Universal Robots PolyScope program: proiectfinal.urp

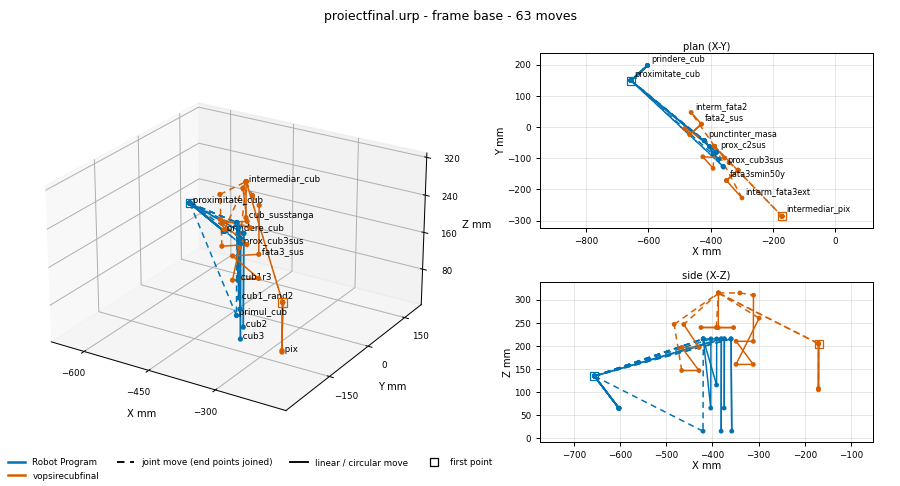
[picture p0: tool path of proiectfinal.urp in frame base, 63 of 63 moves have a stored position in this frame; points joined in program order, loops and branches not executed]
Program testproiectfinal2 (installation=default directory=/programs/usbdisk/final createdIn=3.15.5.106321 lastSavedIn=3.15.6.106324 robotSerialNumber=2021351072)
Calibrated DH parameters: a=[0.000146, -0.006215, -0.392465, 0.000066, 0.00001, 0]; d=[0.089346, 308.112025, -307.666795, -0.334946, 0.094852, 0.082573]; alpha=[1.570365, -0.001381, 0.017393, 1.570287, -1.570555, 0]; deltaTheta=[0.000031, -1.556209, 1.575918, -0.019781, 0.000038, 0.000088]
Robot Program (runOnlyOnce=false)
  MoveJ speed 60 deg/s, acceleration 80 deg/s^2 (useActiveTCP=false) tcp=Palet
    Waypoint proximitate_cub: TCP in base x=-655.658 y=149.782 z=135.002 mm, rx=1.0761 ry=2.3886 rz=1.0065 rad; joints [-7.715, -31.545, 17.047, -40.87, -122.454, -38.841] deg; flange x=-782.032 y=40.366 z=298.765 mm, rx=1.0761 ry=2.3886 rz=1.0065 rad
  MoveL speed 250 mm/s, acceleration 1200 mm/s^2 (useActiveTCP=true) feature=Base
    Waypoint prindere_cub: TCP in base x=-602.576 y=198.07 z=65.356 mm, rx=1.0761 ry=2.3886 rz=1.0065 rad; joints [-11.8, -45.21, 53.1, -65.52, -124.71, -42.93] deg; flange x=-728.95 y=88.654 z=229.118 mm, rx=1.0761 ry=2.3886 rz=1.0065 rad
    Wait Sleep waitTime=0.5
    'G40'
    URCap RG Grip (OnRobot, OnRobot A/S) dataModel(rg-target-force=40.0, rg-target-width=0.04, Variable(key=on_return, variable(name=on_return)))
  MoveL speed 250 mm/s, acceleration 1200 mm/s^2 (useActiveTCP=true) feature=Base
    Waypoint proximitate_cub: TCP in base x=-655.658 y=149.782 z=135.002 mm, rx=1.0761 ry=2.3886 rz=1.0065 rad; joints [-7.715, -31.545, 17.047, -40.87, -122.454, -38.841] deg; flange x=-782.032 y=40.366 z=298.765 mm, rx=1.0761 ry=2.3886 rz=1.0065 rad
  MoveJ speed 60 deg/s, acceleration 80 deg/s^2 (useActiveTCP=true)
    Waypoint punctinter_masa: TCP in base x=-419.876 y=-42.977 z=215.649 mm, rx=2.9437 ry=1.0488 rz=-0.0163 rad; joints [-9.726, -100.905, 97.2, -86.353, -88.88, 41.054] deg; flange x=-418.643 y=-40.621 z=449.643 mm, rx=2.9437 ry=1.0488 rz=-0.0163 rad
  MoveJ speed 60 deg/s, acceleration 80 deg/s^2 (useActiveTCP=true)
    Waypoint primul_cub: TCP in base x=-420.36 y=-43.654 z=15.65 mm, rx=2.9437 ry=1.0488 rz=-0.0163 rad; joints [-9.62, -94.93, 122.37, -117.5, -88.88, 41.16] deg; flange x=-419.127 y=-41.298 z=249.645 mm, rx=2.9437 ry=1.0488 rz=-0.0163 rad
    Wait Sleep waitTime=0.5
    'G80'
    URCap RG Grip (OnRobot, OnRobot A/S) dataModel(rg-target-force=40.0, rg-target-width=0.08)
  MoveJ speed 60 deg/s, acceleration 80 deg/s^2 (useActiveTCP=true)
    Waypoint proximitate_cub: TCP in base x=-655.658 y=149.782 z=135.002 mm, rx=1.0761 ry=2.3886 rz=1.0065 rad; joints [-7.715, -31.545, 17.047, -40.87, -122.454, -38.841] deg; flange x=-782.032 y=40.366 z=298.765 mm, rx=1.0761 ry=2.3886 rz=1.0065 rad
  MoveL speed 250 mm/s, acceleration 1200 mm/s^2 (useActiveTCP=true) feature=Base
    Waypoint prindere_cub: TCP in base x=-602.576 y=198.07 z=65.356 mm, rx=1.0761 ry=2.3886 rz=1.0065 rad; joints [-11.8, -45.21, 53.1, -65.52, -124.71, -42.93] deg; flange x=-728.95 y=88.654 z=229.118 mm, rx=1.0761 ry=2.3886 rz=1.0065 rad
    Wait Sleep waitTime=0.5
    'G40'
    URCap RG Grip (OnRobot, OnRobot A/S) dataModel(rg-target-force=40.0, rg-target-width=0.04)
  MoveJ speed 60 deg/s, acceleration 80 deg/s^2 (useActiveTCP=true)
    Waypoint proximitate_cub: TCP in base x=-655.658 y=149.782 z=135.002 mm, rx=1.0761 ry=2.3886 rz=1.0065 rad; joints [-7.715, -31.545, 17.047, -40.87, -122.454, -38.841] deg; flange x=-782.032 y=40.366 z=298.765 mm, rx=1.0761 ry=2.3886 rz=1.0065 rad
  MoveL speed 250 mm/s, acceleration 1200 mm/s^2 (useActiveTCP=true) feature=Base
    Waypoint prox_c2sus: TCP in base x=-380.694 y=-80.38 z=215.695 mm, rx=2.9437 ry=1.0488 rz=-0.0163 rad; joints [-4.992, -105.625, 100.759, -85.284, -88.888, 45.789] deg; flange x=-379.461 y=-78.023 z=449.69 mm, rx=2.9437 ry=1.0488 rz=-0.0163 rad
  MoveL speed 250 mm/s, acceleration 1200 mm/s^2 (useActiveTCP=true) feature=Base
    Waypoint cub2: TCP in base x=-381.178 y=-81.057 z=15.697 mm, rx=2.9437 ry=1.0488 rz=-0.0163 rad; joints [-4.881, -99.963, 126.628, -116.816, -88.889, 45.899] deg; flange x=-379.945 y=-78.7 z=249.691 mm, rx=2.9437 ry=1.0488 rz=-0.0163 rad
    Wait Sleep waitTime=0.5
    'G80'
    URCap RG Grip (OnRobot, OnRobot A/S) dataModel(rg-target-force=40.0, rg-target-width=0.08)
  MoveL speed 250 mm/s, acceleration 1200 mm/s^2 (useActiveTCP=true) feature=Base
    Waypoint prox_cub2: TCP in base x=-380.694 y=-80.38 z=215.695 mm, rx=2.9437 ry=1.0488 rz=-0.0163 rad; joints [-4.992, -105.625, 100.759, -85.284, -88.888, 45.789] deg; flange x=-379.461 y=-78.023 z=449.69 mm, rx=2.9437 ry=1.0488 rz=-0.0163 rad
  MoveJ speed 60 deg/s, acceleration 80 deg/s^2 (useActiveTCP=true)
    Waypoint proximitate_cub: TCP in base x=-655.658 y=149.782 z=135.002 mm, rx=1.0761 ry=2.3886 rz=1.0065 rad; joints [-7.715, -31.545, 17.047, -40.87, -122.454, -38.841] deg; flange x=-782.032 y=40.366 z=298.765 mm, rx=1.0761 ry=2.3886 rz=1.0065 rad
  MoveL speed 250 mm/s, acceleration 1200 mm/s^2 (useActiveTCP=true) feature=Base
    Waypoint prindere_cub: TCP in base x=-602.576 y=198.07 z=65.356 mm, rx=1.0761 ry=2.3886 rz=1.0065 rad; joints [-11.8, -45.21, 53.1, -65.52, -124.71, -42.93] deg; flange x=-728.95 y=88.654 z=229.118 mm, rx=1.0761 ry=2.3886 rz=1.0065 rad
    Wait Sleep waitTime=0.5
    'G40'
    URCap RG Grip (OnRobot, OnRobot A/S) dataModel(rg-target-force=40.0, rg-target-width=0.04)
  MoveJ speed 60 deg/s, acceleration 80 deg/s^2 (useActiveTCP=true)
    Waypoint proximitate_cub: TCP in base x=-655.658 y=149.782 z=135.002 mm, rx=1.0761 ry=2.3886 rz=1.0065 rad; joints [-7.715, -31.545, 17.047, -40.87, -122.454, -38.841] deg; flange x=-782.032 y=40.366 z=298.765 mm, rx=1.0761 ry=2.3886 rz=1.0065 rad
  MoveJ speed 60 deg/s, acceleration 80 deg/s^2 (useActiveTCP=true)
    Waypoint prox_cub3sus: TCP in base x=-359.676 y=-125.655 z=215.741 mm, rx=2.9437 ry=1.0488 rz=-0.0163 rad; joints [2.001, -106.845, 101.634, -85.073, -88.915, 52.783] deg; flange x=-358.443 y=-123.298 z=449.736 mm, rx=2.9437 ry=1.0488 rz=-0.0163 rad
  MoveL speed 250 mm/s, acceleration 1200 mm/s^2 (useActiveTCP=true) feature=Base
    Waypoint cub3: TCP in base x=-358.165 y=-128.509 z=15.708 mm, rx=2.9439 ry=1.0486 rz=-0.0162 rad; joints [2.174, -101.579, 127.644, -116.344, -87.985, 53.434] deg; flange x=-356.947 y=-126.168 z=249.703 mm, rx=2.9439 ry=1.0486 rz=-0.0162 rad
    Wait Sleep waitTime=0.5
    'G80'
    URCap RG Grip (OnRobot, OnRobot A/S) dataModel(rg-target-force=40.0, rg-target-width=0.08)
  MoveL speed 250 mm/s, acceleration 1200 mm/s^2 (useActiveTCP=true) feature=Base
    Waypoint prox_cub3: TCP in base x=-359.676 y=-125.655 z=215.741 mm, rx=2.9437 ry=1.0488 rz=-0.0163 rad; joints [2.001, -106.845, 101.634, -85.073, -88.915, 52.783] deg; flange x=-358.443 y=-123.298 z=449.736 mm, rx=2.9437 ry=1.0488 rz=-0.0163 rad
  MoveJ speed 60 deg/s, acceleration 80 deg/s^2 (useActiveTCP=true)
    Waypoint proximitate_cub: TCP in base x=-655.658 y=149.782 z=135.002 mm, rx=1.0761 ry=2.3886 rz=1.0065 rad; joints [-7.715, -31.545, 17.047, -40.87, -122.454, -38.841] deg; flange x=-782.032 y=40.366 z=298.765 mm, rx=1.0761 ry=2.3886 rz=1.0065 rad
  MoveL speed 250 mm/s, acceleration 1200 mm/s^2 (useActiveTCP=true) feature=Base
    Waypoint prindere_cub: TCP in base x=-602.576 y=198.07 z=65.356 mm, rx=1.0761 ry=2.3886 rz=1.0065 rad; joints [-11.8, -45.21, 53.1, -65.52, -124.71, -42.93] deg; flange x=-728.95 y=88.654 z=229.118 mm, rx=1.0761 ry=2.3886 rz=1.0065 rad
    Wait Sleep waitTime=0.5
    'G40'
    URCap RG Grip (OnRobot, OnRobot A/S) dataModel(rg-target-force=40.0, rg-target-width=0.04)
  MoveL speed 250 mm/s, acceleration 1200 mm/s^2 (useActiveTCP=true) feature=Base
    Waypoint proximitate_cub: TCP in base x=-655.658 y=149.782 z=135.002 mm, rx=1.0761 ry=2.3886 rz=1.0065 rad; joints [-7.715, -31.545, 17.047, -40.87, -122.454, -38.841] deg; flange x=-782.032 y=40.366 z=298.765 mm, rx=1.0761 ry=2.3886 rz=1.0065 rad
  MoveJ speed 60 deg/s, acceleration 80 deg/s^2 (useActiveTCP=true)
    Waypoint punctinter_masa: TCP in base x=-419.876 y=-42.977 z=215.649 mm, rx=2.9437 ry=1.0488 rz=-0.0163 rad; joints [-9.726, -100.905, 97.2, -86.353, -88.88, 41.054] deg; flange x=-418.643 y=-40.621 z=449.643 mm, rx=2.9437 ry=1.0488 rz=-0.0163 rad
  MoveL speed 250 mm/s, acceleration 1200 mm/s^2 (useActiveTCP=true) feature=Base
    Waypoint cub1_rand2: TCP in base x=-403.648 y=-62.186 z=65.673 mm, rx=2.9437 ry=1.0488 rz=-0.0163 rad; joints [-7.34, -100.148, 118.843, -108.8, -88.883, 43.44] deg; flange x=-402.415 y=-59.83 z=299.668 mm, rx=2.9437 ry=1.0488 rz=-0.0163 rad
    Wait Sleep waitTime=0.5
    'G80'
    URCap RG Grip (OnRobot, OnRobot A/S) dataModel(rg-target-force=40.0, rg-target-width=0.08)
  MoveL speed 250 mm/s, acceleration 1200 mm/s^2 (useActiveTCP=true) feature=Base
    Waypoint ridicare_cub1r2: TCP in base x=-403.285 y=-61.678 z=215.672 mm, rx=2.9437 ry=1.0488 rz=-0.0163 rad; joints [-7.421, -102.916, 98.768, -85.955, -88.883, 43.359] deg; flange x=-402.052 y=-59.322 z=449.667 mm, rx=2.9437 ry=1.0488 rz=-0.0163 rad
  MoveJ speed 60 deg/s, acceleration 80 deg/s^2 (useActiveTCP=true)
    Waypoint proximitate_cub: TCP in base x=-655.658 y=149.782 z=135.002 mm, rx=1.0761 ry=2.3886 rz=1.0065 rad; joints [-7.715, -31.545, 17.047, -40.87, -122.454, -38.841] deg; flange x=-782.032 y=40.366 z=298.765 mm, rx=1.0761 ry=2.3886 rz=1.0065 rad
  MoveL speed 250 mm/s, acceleration 1200 mm/s^2 (useActiveTCP=true) feature=Base
    Waypoint prindere_cub: TCP in base x=-602.576 y=198.07 z=65.356 mm, rx=1.0761 ry=2.3886 rz=1.0065 rad; joints [-11.8, -45.21, 53.1, -65.52, -124.71, -42.93] deg; flange x=-728.95 y=88.654 z=229.118 mm, rx=1.0761 ry=2.3886 rz=1.0065 rad
    Wait Sleep waitTime=0.5
    'G40'
    URCap RG Grip (OnRobot, OnRobot A/S) dataModel(rg-target-force=40.0, rg-target-width=0.04)
  MoveL speed 250 mm/s, acceleration 1200 mm/s^2 (useActiveTCP=true) feature=Base
    Waypoint proximitate_cub: TCP in base x=-655.658 y=149.782 z=135.002 mm, rx=1.0761 ry=2.3886 rz=1.0065 rad; joints [-7.715, -31.545, 17.047, -40.87, -122.454, -38.841] deg; flange x=-782.032 y=40.366 z=298.765 mm, rx=1.0761 ry=2.3886 rz=1.0065 rad
  MoveJ speed 60 deg/s, acceleration 80 deg/s^2 (useActiveTCP=true)
    Waypoint punctinter_masa: TCP in base x=-419.876 y=-42.977 z=215.649 mm, rx=2.9437 ry=1.0488 rz=-0.0163 rad; joints [-9.726, -100.905, 97.2, -86.353, -88.88, 41.054] deg; flange x=-418.643 y=-40.621 z=449.643 mm, rx=2.9437 ry=1.0488 rz=-0.0163 rad
  MoveL speed 250 mm/s, acceleration 1200 mm/s^2 (useActiveTCP=true) feature=Base
    Waypoint prox_c2r2sus: TCP in base x=-374.19 y=-103.473 z=215.718 mm, rx=2.9437 ry=1.0488 rz=-0.0163 rad; joints [-1.482, -105.778, 100.88, -85.32, -88.9, 49.299] deg; flange x=-372.957 y=-101.117 z=449.713 mm, rx=2.9437 ry=1.0488 rz=-0.0163 rad
  MoveL speed 250 mm/s, acceleration 1200 mm/s^2 (useActiveTCP=true) feature=Base
    Waypoint cub2_r2: TCP in base x=-374.553 y=-103.981 z=65.719 mm, rx=2.9437 ry=1.0488 rz=-0.0163 rad; joints [-1.402, -103.233, 121.237, -108.224, -88.9, 49.379] deg; flange x=-373.321 y=-101.625 z=299.714 mm, rx=2.9437 ry=1.0488 rz=-0.0163 rad
    Wait Sleep waitTime=0.5
    'G80'
    URCap RG Grip (OnRobot, OnRobot A/S) dataModel(rg-target-force=40.0, rg-target-width=0.08)
  MoveL speed 250 mm/s, acceleration 1200 mm/s^2 (useActiveTCP=true) feature=Base
    Waypoint prox_cub2r2: TCP in base x=-374.19 y=-103.473 z=215.718 mm, rx=2.9437 ry=1.0488 rz=-0.0163 rad; joints [-1.482, -105.778, 100.88, -85.32, -88.9, 49.299] deg; flange x=-372.958 y=-101.117 z=449.713 mm, rx=2.9437 ry=1.0488 rz=-0.0163 rad
  MoveJ speed 60 deg/s, acceleration 80 deg/s^2 (useActiveTCP=true)
    Waypoint proximitate_cub: TCP in base x=-655.658 y=149.782 z=135.002 mm, rx=1.0761 ry=2.3886 rz=1.0065 rad; joints [-7.715, -31.545, 17.047, -40.87, -122.454, -38.841] deg; flange x=-782.032 y=40.366 z=298.765 mm, rx=1.0761 ry=2.3886 rz=1.0065 rad
  MoveL speed 250 mm/s, acceleration 1200 mm/s^2 (useActiveTCP=true) feature=Base
    Waypoint prindere_cub: TCP in base x=-602.576 y=198.07 z=65.356 mm, rx=1.0761 ry=2.3886 rz=1.0065 rad; joints [-11.8, -45.21, 53.1, -65.52, -124.71, -42.93] deg; flange x=-728.95 y=88.654 z=229.118 mm, rx=1.0761 ry=2.3886 rz=1.0065 rad
    Wait Sleep waitTime=0.5
    'G40'
    URCap RG Grip (OnRobot, OnRobot A/S) dataModel(rg-target-force=40.0, rg-target-width=0.04)
  MoveL speed 250 mm/s, acceleration 1200 mm/s^2 (useActiveTCP=true) feature=Base
    Waypoint proximitate_cub: TCP in base x=-655.658 y=149.782 z=135.002 mm, rx=1.0761 ry=2.3886 rz=1.0065 rad; joints [-7.715, -31.545, 17.047, -40.87, -122.454, -38.841] deg; flange x=-782.032 y=40.366 z=298.765 mm, rx=1.0761 ry=2.3886 rz=1.0065 rad
  MoveJ speed 60 deg/s, acceleration 80 deg/s^2 (useActiveTCP=true)
    Waypoint punctinter_masa: TCP in base x=-419.876 y=-42.977 z=215.649 mm, rx=2.9437 ry=1.0488 rz=-0.0163 rad; joints [-9.726, -100.905, 97.2, -86.353, -88.88, 41.054] deg; flange x=-418.643 y=-40.621 z=449.643 mm, rx=2.9437 ry=1.0488 rz=-0.0163 rad
  MoveL speed 250 mm/s, acceleration 1200 mm/s^2 (useActiveTCP=true) feature=Base
    Waypoint cub1r3: TCP in base x=-391.023 y=-85.111 z=115.696 mm, rx=2.9437 ry=1.0488 rz=-0.0163 rad; joints [-4.15, -103.314, 113.748, -100.6, -88.891, 46.631] deg; flange x=-389.79 y=-82.754 z=349.691 mm, rx=2.9437 ry=1.0488 rz=-0.0163 rad
    Wait Sleep waitTime=0.5
    'G80'
    URCap RG Grip (OnRobot, OnRobot A/S) dataModel(rg-target-force=40.0, rg-target-width=0.08)
  MoveL speed 250 mm/s, acceleration 1200 mm/s^2 (useActiveTCP=true) feature=Base
    Waypoint prox_c3r3s: TCP in base x=-390.781 y=-84.772 z=215.695 mm, rx=2.9437 ry=1.0488 rz=-0.0163 rad; joints [-4.203, -104.095, 99.659, -85.73, -88.891, 46.578] deg; flange x=-389.548 y=-82.415 z=449.69 mm, rx=2.9437 ry=1.0488 rz=-0.0163 rad
  Call vopsirecubfinal
SubProgram -> vopsirecubfinal
SubProgram vopsirecubfinal (keepSynchronizedWithDisk=false) programFile=/home/ur/ursim-current/programs/vopsirecubfinal.urp
  MoveJ speed 60 deg/s, acceleration 80 deg/s^2 (useActiveTCP=true)
    Waypoint intermediar_pix: TCP in base x=-170.071 y=-286.315 z=205.284 mm, rx=1.291 ry=2.848 rz=-0.0146 rad; joints [39.36, -114.129, 107.637, -83.618, -89.01, -1.87] deg; flange x=-170.186 y=-282.604 z=439.264 mm, rx=1.291 ry=2.848 rz=-0.0146 rad
  MoveL speed 250 mm/s, acceleration 1200 mm/s^2 (useActiveTCP=true) feature=Base
    Waypoint pix: TCP in base x=-170.313 y=-286.653 z=105.285 mm, rx=1.291 ry=2.848 rz=-0.0146 rad; joints [39.38, -113.83, 122.12, -98.4, -89.01, -1.85] deg; flange x=-170.428 y=-282.942 z=339.265 mm, rx=1.291 ry=2.848 rz=-0.0146 rad
    Wait Sleep waitTime=0.5
    URCap RG Grip (OnRobot, OnRobot A/S) dataModel(rg-target-force=40.0, rg-target-width=0.01)
    'G10'
  MoveJ speed 60 deg/s, acceleration 80 deg/s^2 (useActiveTCP=true)
    Waypoint intermediar_pix: TCP in base x=-170.071 y=-286.315 z=205.284 mm, rx=1.291 ry=2.848 rz=-0.0146 rad; joints [39.36, -114.129, 107.637, -83.618, -89.01, -1.87] deg; flange x=-170.186 y=-282.604 z=439.264 mm, rx=1.291 ry=2.848 rz=-0.0146 rad
  MoveJ speed 60 deg/s, acceleration 80 deg/s^2 (useActiveTCP=true)
    Waypoint intermediar_cub: TCP in base x=-387.106 y=-61.589 z=315.134 mm, rx=1.2835 ry=2.8619 rz=-0.034 rad; joints [-8.293, -102.753, 83.777, -71.093, -88.73, -49.983] deg; flange x=-383.978 y=-56.18 z=549.06 mm, rx=1.2835 ry=2.8619 rz=-0.034 rad
  MoveL speed 250 mm/s, acceleration 1200 mm/s^2 (useActiveTCP=true) feature=Base
    Waypoint cub_susstanga: TCP in base x=-387.287 y=-61.843 z=240.134 mm, rx=1.2835 ry=2.8619 rz=-0.034 rad; joints [-8.25, -105.11, 96.79, -81.75, -88.73, -49.94] deg; flange x=-384.16 y=-56.434 z=474.061 mm, rx=1.2835 ry=2.8619 rz=-0.034 rad
  MoveL speed 250 mm/s, acceleration 1200 mm/s^2 (useActiveTCP=true) feature=Base
    Waypoint cub_susdreapta: TCP in base x=-354.105 y=-99.246 z=240.181 mm, rx=1.2835 ry=2.8619 rz=-0.034 rad; joints [-2.814, -108.653, 99.227, -80.764, -88.742, -44.503] deg; flange x=-350.978 y=-93.837 z=474.107 mm, rx=1.2835 ry=2.8619 rz=-0.034 rad
  MoveL speed 250 mm/s, acceleration 1200 mm/s^2 (useActiveTCP=true) feature=Base
    Waypoint diagstangjos: TCP in base x=-424.69 y=-95.025 z=240.337 mm, rx=1.2835 ry=2.8619 rz=-0.034 rad; joints [-2.918, -99.183, 92.225, -83.229, -88.742, -44.606] deg; flange x=-421.562 y=-89.615 z=474.264 mm, rx=1.2835 ry=2.8619 rz=-0.034 rad
  MoveL speed 250 mm/s, acceleration 1200 mm/s^2 (useActiveTCP=true) feature=Base
    Waypoint cub_dreaptajos: TCP in base x=-391.508 y=-132.427 z=240.384 mm, rx=1.2835 ry=2.8619 rz=-0.034 rad; joints [2.359, -102.313, 94.738, -82.728, -88.765, -39.328] deg; flange x=-388.38 y=-127.018 z=474.31 mm, rx=1.2835 ry=2.8619 rz=-0.034 rad
  MoveJ speed 60 deg/s, acceleration 80 deg/s^2 (useActiveTCP=true)
    Waypoint intermediar_cub: TCP in base x=-387.106 y=-61.589 z=315.134 mm, rx=1.2835 ry=2.8619 rz=-0.034 rad; joints [-8.293, -102.753, 83.777, -71.093, -88.73, -49.983] deg; flange x=-383.978 y=-56.18 z=549.06 mm, rx=1.2835 ry=2.8619 rz=-0.034 rad
  MoveJ speed 60 deg/s, acceleration 80 deg/s^2 (useActiveTCP=true)
    Waypoint interm_latdrcub: TCP in base x=-340.651 y=-113.953 z=315.198 mm, rx=1.2835 ry=2.8619 rz=-0.034 rad; joints [-0.408, -107.27, 86.983, -69.955, -88.751, -42.096] deg; flange x=-337.523 y=-108.544 z=549.125 mm, rx=1.2835 ry=2.8619 rz=-0.034 rad
  MoveJ speed 60 deg/s, acceleration 80 deg/s^2 (useActiveTCP=true)
    Waypoint interm_fata3: TCP in base x=-311.097 y=-137.967 z=310.289 mm, rx=-0.1394 ry=-2.5859 rz=-0.5323 rad; joints [36.655, -116.066, 104.459, -87.091, -125.726, -49.98] deg; flange x=-205.123 y=-228.798 z=498.118 mm, rx=-0.1394 ry=-2.5859 rz=-0.5323 rad
  MoveL speed 250 mm/s, acceleration 1200 mm/s^2 (useActiveTCP=true) feature=Base
    Waypoint fata3_sus: TCP in base x=-311.331 y=-138.32 z=210.278 mm, rx=-0.1394 ry=-2.586 rz=-0.5323 rad; joints [36.68, -117.15, 119.7, -101.23, -125.726, -49.95] deg; flange x=-205.363 y=-229.14 z=398.116 mm, rx=-0.1394 ry=-2.586 rz=-0.5323 rad
  MoveL speed 250 mm/s, acceleration 1200 mm/s^2 (useActiveTCP=true) feature=Base
    Waypoint fata3smin50y: TCP in base x=-348.733 y=-171.502 z=210.481 mm, rx=-0.1394 ry=-2.586 rz=-0.5323 rad; joints [37.395, -109.418, 115.134, -103.887, -125.831, -49.078] deg; flange x=-242.766 y=-262.322 z=398.319 mm, rx=-0.1394 ry=-2.586 rz=-0.5323 rad
  MoveL speed 250 mm/s, acceleration 1200 mm/s^2 (useActiveTCP=true) feature=Base
    Waypoint diag: TCP in base x=-311.452 y=-138.489 z=160.278 mm, rx=-0.1394 ry=-2.586 rz=-0.5323 rad; joints [36.692, -116.21, 126.574, -109.035, -125.728, -49.935] deg; flange x=-205.484 y=-229.309 z=348.116 mm, rx=-0.1394 ry=-2.586 rz=-0.5323 rad
  MoveL speed 250 mm/s, acceleration 1200 mm/s^2 (useActiveTCP=true) feature=Base
    Waypoint fata3josmin50y: TCP in base x=-348.854 y=-171.671 z=160.481 mm, rx=-0.1394 ry=-2.586 rz=-0.5323 rad; joints [37.405, -108.1, 121.695, -111.758, -125.832, -49.066] deg; flange x=-242.887 y=-262.491 z=348.319 mm, rx=-0.1394 ry=-2.586 rz=-0.5323 rad
  MoveL speed 250 mm/s, acceleration 1200 mm/s^2 (useActiveTCP=true) feature=Base
    Waypoint interm_fata3ext: TCP in base x=-298.839 y=-227.436 z=260.55 mm, rx=-0.1394 ry=-2.586 rz=-0.5323 rad; joints [49.496, -106.173, 103.501, -86.61, -126.623, -34.094] deg; flange x=-192.872 y=-318.256 z=448.388 mm, rx=-0.1394 ry=-2.586 rz=-0.5323 rad
  MoveJ speed 60 deg/s, acceleration 80 deg/s^2 (useActiveTCP=true)
    Waypoint intermediar_cub: TCP in base x=-387.106 y=-61.589 z=315.134 mm, rx=1.2835 ry=2.8619 rz=-0.034 rad; joints [-8.293, -102.753, 83.777, -71.093, -88.73, -49.983] deg; flange x=-383.978 y=-56.18 z=549.06 mm, rx=1.2835 ry=2.8619 rz=-0.034 rad
  MoveJ speed 60 deg/s, acceleration 80 deg/s^2 (useActiveTCP=true)
    Waypoint interm_fata2: TCP in base x=-462.134 y=47.249 z=246.923 mm, rx=1.5541 ry=1.7177 rz=-0.4294 rad; joints [-35.631, -69.065, 63.951, -39.612, -67.495, -50.842] deg; flange x=-533.143 y=209.077 z=400.318 mm, rx=1.5541 ry=1.7177 rz=-0.4294 rad
  MoveL speed 250 mm/s, acceleration 1200 mm/s^2 (useActiveTCP=true) feature=Base
    Waypoint fata2_sus: TCP in base x=-429.073 y=9.677 z=196.969 mm, rx=1.5541 ry=1.7177 rz=-0.4294 rad; joints [-34.48, -75.75, 80.19, -49.51, -66.68, -49.96] deg; flange x=-500.082 y=171.505 z=350.364 mm, rx=1.5541 ry=1.7177 rz=-0.4294 rad
  MoveL speed 250 mm/s, acceleration 1200 mm/s^2 (useActiveTCP=true) feature=Base
    Waypoint fata2susmin50y: TCP in base x=-466.475 y=-23.504 z=197.172 mm, rx=1.5541 ry=1.7177 rz=-0.4294 rad; joints [-29.692, -72.801, 76.621, -50.493, -63.345, -46.169] deg; flange x=-537.484 y=138.324 z=350.567 mm, rx=1.5541 ry=1.7177 rz=-0.4294 rad
  MoveL speed 250 mm/s, acceleration 1200 mm/s^2 (useActiveTCP=true) feature=Base
    Waypoint diag2: TCP in base x=-429.194 y=9.508 z=146.97 mm, rx=1.5541 ry=1.7177 rz=-0.4294 rad; joints [-34.459, -74.801, 86.357, -56.633, -66.665, -49.944] deg; flange x=-500.203 y=171.336 z=300.365 mm, rx=1.5541 ry=1.7177 rz=-0.4294 rad
  MoveL speed 250 mm/s, acceleration 1200 mm/s^2 (useActiveTCP=true) feature=Base
    Waypoint fata2josmin50y: TCP in base x=-466.596 y=-23.673 z=147.173 mm, rx=1.5541 ry=1.7177 rz=-0.4294 rad; joints [-29.671, -71.916, 82.814, -57.578, -63.331, -46.152] deg; flange x=-537.605 y=138.154 z=300.568 mm, rx=1.5541 ry=1.7177 rz=-0.4294 rad
  MoveJ speed 60 deg/s, acceleration 80 deg/s^2 (useActiveTCP=true)
    Waypoint fata2_intermext: TCP in base x=-482.945 y=-4.634 z=247.149 mm, rx=1.5541 ry=1.7177 rz=-0.4294 rad; joints [-30.467, -69.526, 64.844, -41.712, -63.878, -46.796] deg; flange x=-553.954 y=157.194 z=400.544 mm, rx=1.5541 ry=1.7177 rz=-0.4294 rad
  MoveJ speed 60 deg/s, acceleration 80 deg/s^2 (useActiveTCP=true)
    Waypoint intermediar_cub: TCP in base x=-387.106 y=-61.589 z=315.134 mm, rx=1.2835 ry=2.8619 rz=-0.034 rad; joints [-8.293, -102.753, 83.777, -71.093, -88.73, -49.983] deg; flange x=-383.978 y=-56.18 z=549.06 mm, rx=1.2835 ry=2.8619 rz=-0.034 rad
  MoveJ speed 60 deg/s, acceleration 80 deg/s^2 (useActiveTCP=true)
    Waypoint intermediar_pix: TCP in base x=-170.071 y=-286.315 z=205.284 mm, rx=1.291 ry=2.848 rz=-0.0146 rad; joints [39.36, -114.129, 107.637, -83.618, -89.01, -1.87] deg; flange x=-170.186 y=-282.604 z=439.264 mm, rx=1.291 ry=2.848 rz=-0.0146 rad
  MoveL speed 250 mm/s, acceleration 1200 mm/s^2 (useActiveTCP=true) feature=Base
    Waypoint Waypoint_1: TCP in base x=-170.325 y=-286.651 z=108.284 mm, rx=1.2911 ry=2.848 rz=-0.0148 rad; joints [39.139, -113.999, 121.511, -97.612, -87.981, -1.942] deg; flange x=-170.411 y=-282.927 z=342.264 mm, rx=1.2911 ry=2.848 rz=-0.0148 rad
    Wait Sleep waitTime=0.5
    'G40'
    URCap RG Grip (OnRobot, OnRobot A/S) dataModel(rg-target-force=40.0, rg-target-width=0.04)
  MoveL speed 250 mm/s, acceleration 1200 mm/s^2 (useActiveTCP=true) feature=Base
    Waypoint intermediar_pix: TCP in base x=-170.071 y=-286.315 z=205.284 mm, rx=1.291 ry=2.848 rz=-0.0146 rad; joints [39.36, -114.129, 107.637, -83.618, -89.01, -1.87] deg; flange x=-170.186 y=-282.604 z=439.264 mm, rx=1.291 ry=2.848 rz=-0.0146 rad
